// TIA Portal project "Ejercicio3_GruaCiclos" (V15.1)

(* hardware
DEVICE "S7-1200 station_1"  S7-1200 Station
   slot 0: "Rack_0"  S7-1200 Rack  Rack  V1.0
   slot 1: "PLC_1"  CPU 1214C AC/DC/Rly  6ES7 214-1BG40-0XB0  V4.2
*)

// ===== PLC "PLC_1"  CPU 1214C AC/DC/Rly =====

VAR_GLOBAL   // PLC tag table "Tabla de variables estándar"
   "Etapa0" AT %M16.0 : Bool;
   "Etapa1" AT %M16.1 : Bool;
   "Etapa2" AT %M16.2 : Bool;
   "Etapa3" AT %M16.3 : Bool;
   "Etapa4" AT %M16.4 : Bool;
   "Etapa5" AT %M16.5 : Bool;
   "Etapa6" AT %M16.6 : Bool;
   "Etapa7" AT %M16.7 : Bool;
   "FC1" AT %I1.0 : Bool;
   "FC2" AT %I1.1 : Bool;
   "FC3" AT %I1.2 : Bool;
   "FC4" AT %I1.3 : Bool;
   "M" AT %I1.4 : Bool;
   "KM_Left" AT %Q1.0 : Bool;
   "KM_Right" AT %Q1.1 : Bool;
   "KM_Up" AT %Q0.2 : Bool;
   "KM_Down" AT %Q0.3 : Bool;
END_VAR

// folder: System blocks/Program resources

DATA_BLOCK "Temporizador1"   // DB1
{ S7_Optimized_Access := 'TRUE' }
AUTHOR : Simatic
FAMILY : IEC
NAME : IEC_TMR
VERSION : 1.0
// stored: InstanceOfName IEC_TIMER
"IEC_TIMER"
BEGIN
END_DATA_BLOCK

// folder: (top level)

ORGANIZATION_BLOCK "Main"   // OB1, LAD, ProgramCycle
TITLE = "Main Program Sweep (Cycle)"
{ S7_Optimized_Access := 'TRUE' }
VERSION : 0.1
   VAR_INPUT
      Initial_Call : Bool;   // Initial call of this OB
      Remanence : Bool;   // =True, if remanent data are available
   END_VAR
BEGIN

REGION Network 1
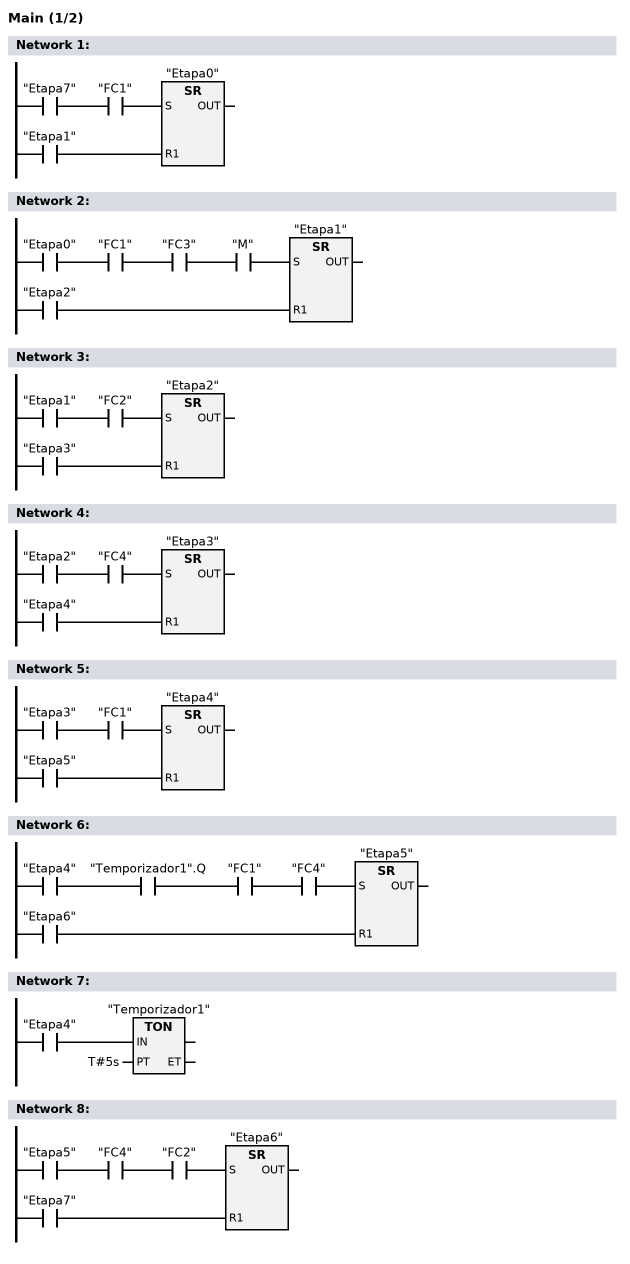
   RUNG wire#powerrail
      Contact( "Etapa7" )
      Contact( "FC1" )
      S_SR(operand := "Etapa0", r1 := wire#w1)
   END_RUNG
   RUNG wire#powerrail
      Contact( "Etapa1" )
   END_RUNG wire#w1
   // the same network as SCL:
   IF "Etapa7" AND "FC1" THEN
       "Etapa0" := TRUE;   // SR flip-flop
   END_IF;
   IF "Etapa1" THEN "Etapa0" := FALSE; END_IF;
END_REGION

REGION Network 2
   RUNG wire#powerrail
      Contact( "Etapa0" )
      Contact( "FC1" )
      Contact( "FC3" )
      Contact( "M" )
      S_SR(operand := "Etapa1", r1 := wire#w1)
   END_RUNG
   RUNG wire#powerrail
      Contact( "Etapa2" )
   END_RUNG wire#w1
   // the same network as SCL:
   IF "Etapa0" AND "FC1" AND "FC3" AND "M" THEN
       "Etapa1" := TRUE;   // SR flip-flop
   END_IF;
   IF "Etapa2" THEN "Etapa1" := FALSE; END_IF;
END_REGION

REGION Network 3
   RUNG wire#powerrail
      Contact( "Etapa1" )
      Contact( "FC2" )
      S_SR(operand := "Etapa2", r1 := wire#w1)
   END_RUNG
   RUNG wire#powerrail
      Contact( "Etapa3" )
   END_RUNG wire#w1
   // the same network as SCL:
   IF "Etapa1" AND "FC2" THEN
       "Etapa2" := TRUE;   // SR flip-flop
   END_IF;
   IF "Etapa3" THEN "Etapa2" := FALSE; END_IF;
END_REGION

REGION Network 4
   RUNG wire#powerrail
      Contact( "Etapa2" )
      Contact( "FC4" )
      S_SR(operand := "Etapa3", r1 := wire#w1)
   END_RUNG
   RUNG wire#powerrail
      Contact( "Etapa4" )
   END_RUNG wire#w1
   // the same network as SCL:
   IF "Etapa2" AND "FC4" THEN
       "Etapa3" := TRUE;   // SR flip-flop
   END_IF;
   IF "Etapa4" THEN "Etapa3" := FALSE; END_IF;
END_REGION

REGION Network 5
   RUNG wire#powerrail
      Contact( "Etapa3" )
      Contact( "FC1" )
      S_SR(operand := "Etapa4", r1 := wire#w1)
   END_RUNG
   RUNG wire#powerrail
      Contact( "Etapa5" )
   END_RUNG wire#w1
   // the same network as SCL:
   IF "Etapa3" AND "FC1" THEN
       "Etapa4" := TRUE;   // SR flip-flop
   END_IF;
   IF "Etapa5" THEN "Etapa4" := FALSE; END_IF;
END_REGION

REGION Network 6
   RUNG wire#powerrail
      Contact( "Etapa4" )
      Contact( "Temporizador1".Q )
      Contact( "FC1" )
      Contact( "FC4" )
      S_SR(operand := "Etapa5", r1 := wire#w1)
   END_RUNG
   RUNG wire#powerrail
      Contact( "Etapa6" )
   END_RUNG wire#w1
   // the same network as SCL:
   IF "Etapa4" AND "Temporizador1".Q AND "FC1" AND "FC4" THEN
       "Etapa5" := TRUE;   // SR flip-flop
   END_IF;
   IF "Etapa6" THEN "Etapa5" := FALSE; END_IF;
END_REGION

REGION Network 7
   "Temporizador1".TON(IN := "Etapa4", PT := T#5s);
END_REGION

REGION Network 8
   RUNG wire#powerrail
      Contact( "Etapa5" )
      Contact( "FC4" )
      Contact( "FC2" )
      S_SR(operand := "Etapa6", r1 := wire#w1)
   END_RUNG
   RUNG wire#powerrail
      Contact( "Etapa7" )
   END_RUNG wire#w1
   // the same network as SCL:
   IF "Etapa5" AND "FC4" AND "FC2" THEN
       "Etapa6" := TRUE;   // SR flip-flop
   END_IF;
   IF "Etapa7" THEN "Etapa6" := FALSE; END_IF;
END_REGION

REGION Network 9
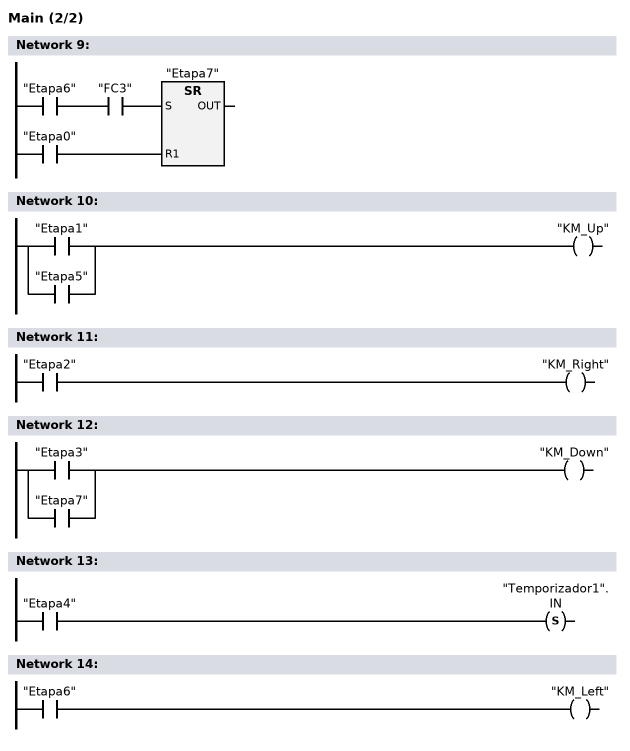
   RUNG wire#powerrail
      Contact( "Etapa6" )
      Contact( "FC3" )
      S_SR(operand := "Etapa7", r1 := wire#w1)
   END_RUNG
   RUNG wire#powerrail
      Contact( "Etapa0" )
   END_RUNG wire#w1
   // the same network as SCL:
   IF "Etapa6" AND "FC3" THEN
       "Etapa7" := TRUE;   // SR flip-flop
   END_IF;
   IF "Etapa0" THEN "Etapa7" := FALSE; END_IF;
END_REGION

REGION Network 10
   RUNG wire#powerrail
      Contact( "Etapa1" )
      wire#w1
      Coil( "KM_Up" )
   END_RUNG
   RUNG wire#powerrail
      Contact( "Etapa5" )
   END_RUNG wire#w1
   // the same network as SCL:
   "KM_Up" := "Etapa1" OR "Etapa5";
END_REGION

REGION Network 11
   RUNG wire#powerrail
      Contact( "Etapa2" )
      Coil( "KM_Right" )
   END_RUNG
   // the same network as SCL:
   "KM_Right" := "Etapa2";
END_REGION

REGION Network 12
   RUNG wire#powerrail
      Contact( "Etapa3" )
      wire#w1
      Coil( "KM_Down" )
   END_RUNG
   RUNG wire#powerrail
      Contact( "Etapa7" )
   END_RUNG wire#w1
   // the same network as SCL:
   "KM_Down" := "Etapa3" OR "Etapa7";
END_REGION

REGION Network 13
   RUNG wire#powerrail
      Contact( "Etapa4" )
      S_Coil( "Temporizador1".IN )
   END_RUNG
   // the same network as SCL:
   IF "Etapa4" THEN "Temporizador1".IN := TRUE; END_IF;
END_REGION

REGION Network 14
   RUNG wire#powerrail
      Contact( "Etapa6" )
      Coil( "KM_Left" )
   END_RUNG
   // the same network as SCL:
   "KM_Left" := "Etapa6";
END_REGION
END_ORGANIZATION_BLOCK

ORGANIZATION_BLOCK "Startup"   // OB100, LAD, Startup
TITLE = "Complete Restart"
{ S7_Optimized_Access := 'TRUE' }
VERSION : 0.1
   VAR_INPUT
      LostRetentive : Bool;   // True if retentive data are lost
      LostRTC : Bool;   // True if date and time are lost
   END_VAR
BEGIN

REGION Network 1
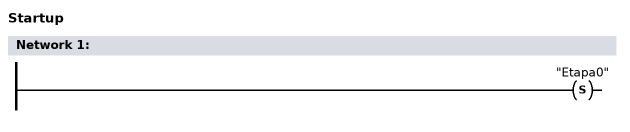
   RUNG wire#powerrail
      S_Coil( "Etapa0" )
   END_RUNG
   // the same network as SCL:
   "Etapa0" := TRUE;
END_REGION
END_ORGANIZATION_BLOCK